FUNCTION_BLOCK FB_SEL_WSTRING (* WSTRING Selection *)
  (* Standard: 61499-1-D.1; Classification: Selection Functions *)
  (* Version 0.1, 2001-08-06, JHC, Rockwell Automation, XML version *)
  (* Version 0.0, 2000-01-11, JHC, Rockwell Automation, SRC version *)
  (* Compiler header: package fb.rt.math; *)
  (* Compiler classdef: class FB_SEL_WSTRING extends FBSelectFunction *)
  (* Compiler Java IBM VisualAge 3.0 *)
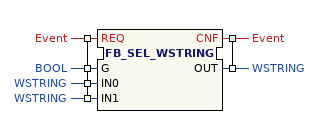
  EVENT_INPUT
    REQ WITH G, IN0, IN1;
  END_EVENT
  EVENT_OUTPUT
    CNF WITH OUT;
  END_EVENT
  VAR_INPUT
    G : BOOL; (* Selector *)
    IN0 : WSTRING; (* Selected when G=0 *)
    IN1 : WSTRING; (* Selected when G=1 *)
  END_VAR
  VAR_OUTPUT
    OUT : WSTRING; (* Selected value *)
  END_VAR
END_FUNCTION_BLOCK
